def draw_auto_center_screen(
    color_image_bgr,
    box,
    stable_frame_count,
    failed_auto_moves,
    total_auto_moves,
):
    draw_auto_text(
        color_image_bgr,
        "AUTO CENTERING BEFORE SCAN",
        30,
        (0, 255, 255),
    )

    draw_auto_text(
        color_image_bgr,
        "S = start scan manually | H = home | C = center reference | Q = quit",
        60,
        (255, 255, 255),
    )

    draw_auto_text(
        color_image_bgr,
        f"Moves: {total_auto_moves}/{AUTO_MAX_TOTAL_MOVES} | Failed: {failed_auto_moves}/{AUTO_MAX_FAILED_MOVES}",
        90,
        (255, 255, 255),
    )

    if box is None:
        draw_auto_text(
            color_image_bgr,
            "No box detected",
            120,
            (0, 0, 255),
        )
        return

    draw_auto_box(color_image_bgr, box)

    offset_x, offset_y = get_auto_box_offset_pixels(box)
    centered_status = "Centered" if is_auto_box_centered(box) else "Moving"

    draw_auto_text(
        color_image_bgr,
        (
            f"Offset X={offset_x}px Y={offset_y}px | "
            f"{centered_status} | Stable {stable_frame_count}/{AUTO_REQUIRED_STABLE_FRAMES}"
        ),
        120,
        (0, 255, 0),
    )


def close_auto_windows():
    for window_name in [AUTO_WINDOW_NAME, AUTO_MASK_WINDOW_NAME]:
        try:
            cv2.destroyWindow(window_name)
        except cv2.error:
            pass


def auto_center_camera_on_box(
    robot,
    rdk,
    pipeline,
    align,
    depth_scale,
    T_tcp_camera,
    T_camera_tcp,
):
    previous_box = None
    stable_frame_count = 0
    failed_auto_moves = 0
    total_auto_moves = 0
    last_auto_move_time = 0.0
    start_time = time.time()
    last_print_time = 0.0

    print("")
    print("=" * 70)
    print("AUTO CENTERING STARTED")
    print("=" * 70)
    print("The robot will center the camera on the detected open box.")
    print("When centered, the code will continue with the reference capture.")
    print("Press S to skip centering and start the scan from the current pose.")
    print("=" * 70)

    while True:
        if time.time() - start_time > AUTO_CENTER_TIMEOUT_SECONDS:
            close_auto_windows()
            raise Exception("Auto centering timed out before the box was centered.")

        depth_frame, color_image_rgb, depth_image = get_aligned_realsense_frame(
            pipeline,
            align,
        )

        if depth_frame is None:
            continue

        color_image_bgr = cv2.cvtColor(color_image_rgb, cv2.COLOR_RGB2BGR)
        box, mask = detect_auto_box(depth_image, depth_scale)

        stable_frame_count, previous_box = update_auto_stability(
            box,
            previous_box,
            stable_frame_count,
        )

        draw_auto_center_screen(
            color_image_bgr,
            box,
            stable_frame_count,
            failed_auto_moves,
            total_auto_moves,
        )

        if box is not None and time.time() - last_print_time > 0.5:
            offset_x, offset_y = get_auto_box_offset_pixels(box)
            print(
                "Auto box:",
                f"center=({box['center_x']}, {box['center_y']}),",
                f"offset=({offset_x}, {offset_y}),",
                f"distance={box['distance_meters']:.2f}m,",
                f"stable={stable_frame_count}/{AUTO_REQUIRED_STABLE_FRAMES}",
            )
            last_print_time = time.time()

        if mask is not None:
            cv2.imshow(AUTO_MASK_WINDOW_NAME, mask)

        cv2.imshow(AUTO_WINDOW_NAME, color_image_bgr)

        key = cv2.waitKey(1) & 0xFF

        if key == ord("q") or key == 27:
            close_auto_windows()
            raise KeyboardInterrupt

        if key == ord("s"):
            print("")
            print("Manual skip selected. Starting scan from current robot pose.")
            close_auto_windows()
            return get_robot_joints_when_ready(robot)

        if key == ord("h"):
            failed_auto_moves = 0
            total_auto_moves = 0
            stable_frame_count = 0
            previous_box = None
            move_robot_to_joints(robot, rdk, HOME_JOINTS, "Home_From_Auto_Center")

        if key == ord("c"):
            failed_auto_moves = 0
            total_auto_moves = 0
            stable_frame_count = 0
            previous_box = None
            move_robot_to_joints(
                robot,
                rdk,
                CENTER_REFERENCE_JOINTS,
                "Center_Reference_From_Auto_Center",
            )

        if box is not None and is_auto_box_centered(box):
            if stable_frame_count >= AUTO_REQUIRED_STABLE_FRAMES:
                print("")
                print("=" * 70)
                print("AUTO CENTERING FINISHED")
                print("=" * 70)
                print("The camera is centered on the box.")
                print("Continuing with reference point cloud capture.")
                print("=" * 70)
                close_auto_windows()
                return get_robot_joints_when_ready(robot)

        if should_auto_center_move(
            box,
            stable_frame_count,
            last_auto_move_time,
            failed_auto_moves,
            total_auto_moves,
        ):
            point_camera = get_auto_box_center_3d(depth_frame, box)

            if point_camera is None:
                print("Auto move skipped. No valid 3D box center.")
                failed_auto_moves += 1
            else:
                actual_joints = move_camera_one_auto_step_to_box_center(
                    robot,
                    rdk,
                    T_tcp_camera,
                    T_camera_tcp,
                    point_camera,
                )

                if actual_joints is None:
                    failed_auto_moves += 1
                else:
                    failed_auto_moves = 0
                    total_auto_moves += 1

            stable_frame_count = 0
            previous_box = None
            last_auto_move_time = time.time()

        if failed_auto_moves >= AUTO_MAX_FAILED_MOVES:
            close_auto_windows()
            raise Exception("Auto centering stopped because too many robot moves failed.")

        if total_auto_moves >= AUTO_MAX_TOTAL_MOVES:
            close_auto_windows()
            raise Exception("Auto centering stopped because the maximum move count was reached.")



# ─────────────────────────────────────────────────────────────────────────────
# MAIN
# ─────────────────────────────────────────────────────────────────────────────

def main():
    OUTPUT_FOLDER.mkdir(parents=True, exist_ok=True)

    rdk = Robolink()
    robot = rdk.ItemUserPick("Select your Doosan M0609 robot", ITEM_TYPE_ROBOT)

    if not robot.Valid():
        raise Exception("No valid robot selected.")

    print("Selected robot:", robot.Name())

    connect_robot(robot, rdk)

    T_tcp_mount = xyzrxryrz_to_numpy(TCP_TO_CAMERA_MOUNT)
    T_mount_optical = xyzrxryrz_to_numpy(CAMERA_MOUNT_TO_OPTICAL)
    T_tcp_camera = T_tcp_mount @ T_mount_optical
    T_camera_tcp = np.linalg.inv(T_tcp_camera)

    print_transform("T_tcp_camera", T_tcp_camera)

    pipeline = None
    combined_point_cloud = o3d.geometry.PointCloud()

    successful_scans = 0
    skipped_scans = 0
    unsafe_scans = 0
    failed_moves = 0

    try:
        (
            pipeline,
            align,
            depth_scale,
            intrinsic_o3d,
            spatial_filter,
            temporal_filter,
            hole_filling_filter,
        ) = start_realsense()

        print("\n" + "=" * 70)
        print("AUTO-CENTERED ADAPTIVE INSIDE-BOX SCANNING STARTED")
        print("=" * 70)
        print("Step 1: Center the camera on the open box.")
        print("Step 2: Capture the reference scan from the centered pose.")
        print("Step 3: Generate adaptive scan poses.")
        print("Step 4: Capture and merge all scans.")
        print("=" * 70)

        if AUTO_CENTER_BEFORE_SCAN:
            center_actual_joints = auto_center_camera_on_box(
                robot,
                rdk,
                pipeline,
                align,
                depth_scale,
                T_tcp_camera,
                T_camera_tcp,
            )
        else:
            center_actual_joints = move_robot_to_joints(
                robot,
                rdk,
                CENTER_REFERENCE_JOINTS,
                "Cabinet_Center_Reference",
            )

        T_base_tcp_center = robodk_mat_to_numpy(robot.SolveFK(center_actual_joints))
        T_base_camera_center = T_base_tcp_center @ T_tcp_camera

        print_transform("T_base_tcp_center", T_base_tcp_center)
        print_transform("T_base_camera_center", T_base_camera_center)

        reference_cloud = capture_stable_pointcloud(
            pipeline,
            align,
            intrinsic_o3d,
            depth_scale,
            spatial_filter,
            temporal_filter,
            hole_filling_filter,
            CAPTURE_FRAMES_PER_POSITION,
        )

        if reference_cloud is None:
            raise Exception("Reference scan failed. No point cloud was captured.")

        print_cloud_bounds("Reference raw camera-frame scan", reference_cloud)
        adaptive_bounds = estimate_camera_cloud_bounds(reference_cloud)

        reference_cloud_cropped = crop_pointcloud_adaptive(
            reference_cloud,
            adaptive_bounds,
        )

        reference_cloud_cropped.transform(T_base_camera_center)
        reference_clean_scan = clean_pointcloud(reference_cloud_cropped)

        if len(reference_clean_scan.points) > 0:
            save_debug_scan("Reference_Center", reference_clean_scan)
            combined_point_cloud += reference_clean_scan
            successful_scans += 1
            print(
                f"Accepted scan {successful_scans}: Reference_Center "
                f"with {len(reference_clean_scan.points):,} cleaned points"
            )
        else:
            print("WARNING: Reference scan became empty after cleaning.")
            skipped_scans += 1

        generated_camera_poses = generate_scan_camera_poses_from_center(
            T_base_camera_center,
            adaptive_bounds,
        )

        for label, T_base_camera_target in generated_camera_poses:
            if label == "Reference_Center":
                continue

            T_base_tcp_target = T_base_camera_target @ T_camera_tcp

            if not is_generated_pose_safe(
                T_base_tcp_target,
                T_base_camera_target,
                label,
            ):
                unsafe_scans += 1
                skipped_scans += 1
                continue

            try:
                actual_joints = move_robot_to_pose(
                    robot,
                    rdk,
                    T_base_tcp_target,
                    label,
                )
            except Exception as error:
                print("")
                print(f"WARNING: Could not move to generated pose {label}.")
                print("Move error:", error)
                failed_moves += 1
                skipped_scans += 1
                continue

            T_base_tcp_actual = robodk_mat_to_numpy(robot.SolveFK(actual_joints))
            T_base_camera_actual = T_base_tcp_actual @ T_tcp_camera

            print_transform(f"T_base_tcp_actual_{label}", T_base_tcp_actual)
            print_transform(f"T_base_camera_actual_{label}", T_base_camera_actual)

            clean_scan = scan_current_position(
                label,
                pipeline,
                align,
                intrinsic_o3d,
                depth_scale,
                spatial_filter,
                temporal_filter,
                hole_filling_filter,
                T_base_camera_actual,
                adaptive_bounds,
            )

            if clean_scan is None:
                skipped_scans += 1
                continue

            combined_point_cloud += clean_scan
            successful_scans += 1

            print(
                f"Accepted scan {successful_scans}: {label} "
                f"with {len(clean_scan.points):,} cleaned points"
            )

    except KeyboardInterrupt:
        print("\nScanning interrupted by user.")

    finally:
        if pipeline is not None:
            pipeline.stop()
            print("\nRealSense stopped.")

        cv2.destroyAllWindows()

        try:
            move_robot_to_joints(
                robot,
                rdk,
                HOME_JOINTS,
                "Home_End",
            )
        except Exception as error:
            print("Could not move robot back to home position:", error)

    print("\n" + "=" * 70)
    print("SCAN SUMMARY")
    print("=" * 70)
    print("Successful scans:", successful_scans)
    print("Skipped scans:", skipped_scans)
    print("Unsafe skipped scans:", unsafe_scans)
    print("Failed robot moves:", failed_moves)
    print("Total merged points before final cleanup:", len(combined_point_cloud.points))
    print_cloud_bounds("Combined point cloud before final cleanup", combined_point_cloud)

    if len(combined_point_cloud.points) == 0:
        raise Exception("No valid point cloud was captured. Combined cloud is empty.")

    combined_point_cloud = clean_pointcloud(combined_point_cloud)
    combined_point_cloud = estimate_normals(combined_point_cloud)

    print("Total merged points after final cleanup:", len(combined_point_cloud.points))
    print_cloud_bounds("Combined point cloud after final cleanup", combined_point_cloud)

    o3d.io.write_point_cloud(str(OUTPUT_CLEAN_FILE), combined_point_cloud)
    print("Saved final merged point cloud to:", OUTPUT_CLEAN_FILE)

    if SHOW_FINAL_CLOUD:
        o3d.visualization.draw_geometries(
            [combined_point_cloud],
            window_name=f"Adaptive Inside Box Point Cloud - {successful_scans} scans",
        )

    print("Done.")


if __name__ == "__main__":
    main()

--- Python program Prog6 ---
import sys
import time
import math

import cv2
import numpy as np
import pyrealsense2 as rs

sys.path.append("C:/RoboDK/Python")

from robodk.robolink import *
from robodk.robomath import TxyzRxyz_2_Pose, Mat


# =============================================================================
# CONFIGURATION
# =============================================================================

RUN_ON_REAL_ROBOT = True

AUTO_MOVE_ENABLED = True
MOVE_TO_CENTER_REFERENCE_ON_START = False

HOME_JOINTS = [270.00, 0.00, 90.00, 180.00, 0.00, 0.00]
CENTER_REFERENCE_JOINTS = [270.01, 0.21, 98.95, 180.00, 6.92, 0.00]

TCP_TO_CAMERA_MOUNT = [0, 0, 55, 0, 0, 0]
CAMERA_MOUNT_TO_OPTICAL = [0, 0, 0, 0, 0, 90]

COLOR_WIDTH = 640
COLOR_HEIGHT = 480
FPS = 30

MIN_DEPTH_METERS = 0.20
MAX_DEPTH_METERS = 3.00
TARGET_DISTANCE_METERS = 0.90

MAX_TRANSLATION_STEP_METERS = 0.025
CENTERING_GAIN = 0.60
DEPTH_GAIN = 0.60

CENTER_TOLERANCE_PIXELS = 25
DISTANCE_TOLERANCE_METERS = 0.05

REQUIRED_STABLE_FRAMES = 8
STABLE_CENTER_TOLERANCE_PIXELS = 12
STABLE_DISTANCE_TOLERANCE_METERS = 0.04
AUTO_MOVE_COOLDOWN_SECONDS = 1.25
MAX_FAILED_AUTO_MOVES = 5

MIN_BOX_AREA = 1200
MIN_BOX_WIDTH = 80
MIN_BOX_HEIGHT = 80

DEPTH_PERCENTILE = 10
DEPTH_FRONT_MARGIN = 0.05
DEPTH_BACK_MARGIN = 0.45

DETECTION_ROI_TOP_RATIO = 0.05
DETECTION_ROI_BOTTOM_RATIO = 0.82
DETECTION_ROI_LEFT_RATIO = 0.02
DETECTION_ROI_RIGHT_RATIO = 0.98

MIN_SAFE_TCP_Z_MM = 120.0
MIN_SAFE_CAMERA_Z_MM = 120.0

SETTLE_TIME = 0.75
MOVE_TIMEOUT_SEC = 30.0
POLL_INTERVAL_SEC = 0.1

WINDOW_NAME = "Automatic Box Centering"
MASK_WINDOW_NAME = "Depth Mask"


# =============================================================================
# MATRIX HELPERS
# =============================================================================

def robodk_mat_to_numpy(mat):
    transform = np.eye(4, dtype=np.float64)

    for row in range(3):
        for col in range(3):
            transform[row, col] = mat[row, col]

        transform[row, 3] = mat[row, 3] / 1000.0

    return transform


def numpy_to_robodk_mat(transform):
    return Mat([
        [
            transform[0, 0],
            transform[0, 1],
            transform[0, 2],
            transform[0, 3] * 1000.0,
        ],
        [
            transform[1, 0],
            transform[1, 1],
            transform[1, 2],
            transform[1, 3] * 1000.0,
        ],
        [
            transform[2, 0],
            transform[2, 1],
            transform[2, 2],
            transform[2, 3] * 1000.0,
        ],
        [0, 0, 0, 1],
    ])


def xyzrxryrz_to_numpy(pose_values):
    pose = TxyzRxyz_2_Pose([
        pose_values[0],
        pose_values[1],
        pose_values[2],
        math.radians(pose_values[3]),
        math.radians(pose_values[4]),
        math.radians(pose_values[5]),
    ])

    return robodk_mat_to_numpy(pose)


def make_local_offset_transform(offset_x, offset_y, offset_z):
    transform = np.eye(4, dtype=np.float64)

    transform[0, 3] = offset_x
    transform[1, 3] = offset_y
    transform[2, 3] = offset_z

    return transform


def joints_to_list(joints_mat):
    try:
        return list(joints_mat.list())
    except Exception:
        try:
            return list(joints_mat)
        except Exception:
            return [joints_mat[index] for index in range(len(joints_mat))]


# =============================================================================
# ROBOT HELPERS
# =============================================================================

def connect_robot(robot, rdk):
    if RUN_ON_REAL_ROBOT:
        rdk.setRunMode(RUNMODE_RUN_ROBOT)

        status = robot.ConnectSafe()
        print("ConnectSafe status:", status)

        if status != ROBOTCOM_READY:
            raise Exception("Robot is not ready. Check RoboDK connection settings.")
    else:
        rdk.setRunMode(RUNMODE_SIMULATE)
        print("Running in RoboDK simulation mode.")


def wait_until_robot_stops(robot, timeout_sec=MOVE_TIMEOUT_SEC):
    start = time.time()

    while True:
        try:
            if not robot.Busy():
                return
        except Exception:
            pass

        if time.time() - start > timeout_sec:
            raise Exception("Timeout waiting for robot to stop.")

        time.sleep(POLL_INTERVAL_SEC)


def get_robot_joints_when_ready(robot, timeout_sec=5.0):
    start = time.time()

    while True:
        try:
            return joints_to_list(robot.Joints())
        except Exception:
            if time.time() - start > timeout_sec:
                raise Exception("Could not read robot joints.")

            time.sleep(POLL_INTERVAL_SEC)


def move_robot_to_joints(robot, rdk, joints, label):
    target = rdk.AddTarget(f"_auto_box_{label}")
    target.setAsJointTarget()
    target.setJoints(joints)

    print("")
    print(f"Moving to {label}: {[round(joint, 2) for joint in joints]}")

    if RUN_ON_REAL_ROBOT:
        rdk.setRunMode(RUNMODE_RUN_ROBOT)
    else:
        rdk.setRunMode(RUNMODE_SIMULATE)

    robot.MoveJ(target, blocking=False)
    wait_until_robot_stops(robot)

    target.Delete()

    print(f"Arrived at {label}. Settling for {SETTLE_TIME:.1f} seconds...")
    time.sleep(SETTLE_TIME)

    return get_robot_joints_when_ready(robot)


def move_robot_to_pose(robot, rdk, T_base_tcp, label):
    target = rdk.AddTarget(f"_auto_box_{label}")
    target_pose = numpy_to_robodk_mat(T_base_tcp)

    target.setPose(target_pose)
    target.setAsCartesianTarget()

    print("")
    print(f"Moving to generated pose: {label}")
    print(f"Target TCP X: {T_base_tcp[0, 3] * 1000.0:.1f} mm")
    print(f"Target TCP Y: {T_base_tcp[1, 3] * 1000.0:.1f} mm")
    print(f"Target TCP Z: {T_base_tcp[2, 3] * 1000.0:.1f} mm")

    if RUN_ON_REAL_ROBOT:
        rdk.setRunMode(RUNMODE_RUN_ROBOT)
    else:
        rdk.setRunMode(RUNMODE_SIMULATE)

    robot.MoveJ(target, blocking=False)
    wait_until_robot_stops(robot)

    target.Delete()

    print(f"Arrived at {label}. Settling for {SETTLE_TIME:.1f} seconds...")
    time.sleep(SETTLE_TIME)

    return get_robot_joints_when_ready(robot)


def is_generated_pose_safe(T_base_tcp, T_base_camera, label):
    tcp_z_mm = T_base_tcp[2, 3] * 1000.0
    camera_z_mm = T_base_camera[2, 3] * 1000.0

    if tcp_z_mm < MIN_SAFE_TCP_Z_MM:
        print("")
        print(f"SKIPPING {label}")
        print(f"Reason: TCP Z is too low: {tcp_z_mm:.1f} mm")
        return False

    if camera_z_mm < MIN_SAFE_CAMERA_Z_MM:
        print("")
        print(f"SKIPPING {label}")
        print(f"Reason: Camera Z is too low: {camera_z_mm:.1f} mm")
        return False

    return True


def calculate_camera_correction(point_camera):
    camera_offset = np.array([
        point_camera[0] * CENTERING_GAIN,
        point_camera[1] * CENTERING_GAIN,
        (point_camera[2] - TARGET_DISTANCE_METERS) * DEPTH_GAIN,
    ])

    offset_size = np.linalg.norm(camera_offset)

    if offset_size > MAX_TRANSLATION_STEP_METERS:
        camera_offset = (
            camera_offset / offset_size
        ) * MAX_TRANSLATION_STEP_METERS

    return camera_offset


def move_camera_one_step_to_box_center(
    robot,
    rdk,
    T_tcp_camera,
    T_camera_tcp,
    point_camera,
):
    actual_joints = get_robot_joints_when_ready(robot)

    T_base_tcp_current = robodk_mat_to_numpy(robot.SolveFK(actual_joints))
    T_base_camera_current = T_base_tcp_current @ T_tcp_camera

    camera_offset = calculate_camera_correction(point_camera)

    T_camera_offset = make_local_offset_transform(
        camera_offset[0],
        camera_offset[1],
        camera_offset[2],
    )

    T_base_camera_target = T_base_camera_current @ T_camera_offset
    T_base_tcp_target = T_base_camera_target @ T_camera_tcp

    print("")
    print("Automatic box-centering movement")
    print("3D box point in camera frame:", np.round(point_camera, 4), "m")
    print("Camera movement step:", np.round(camera_offset, 4), "m")
    print("Current robot joints:", [round(joint, 2) for joint in actual_joints])

    if not is_generated_pose_safe(
        T_base_tcp_target,
        T_base_camera_target,
        "Auto_Box_Center_Step",
    ):
        return None

    try:
        return move_robot_to_pose(
            robot,
            rdk,
            T_base_tcp_target,
            "Auto_Box_Center_Step",
        )
    except Exception as error:
        print("")
        print("Could not move robot to automatic box center step.")
        print("Move error:", error)
        return None


# =============================================================================
# REALSENSE HELPERS
# =============================================================================

def start_realsense():
    print("")
    print("Starting Intel RealSense camera...")

    pipeline = rs.pipeline()
    config = rs.config()

    config.enable_stream(
        rs.stream.color,
        COLOR_WIDTH,
        COLOR_HEIGHT,
        rs.format.bgr8,
        FPS,
    )

    config.enable_stream(
        rs.stream.depth,
        COLOR_WIDTH,
        COLOR_HEIGHT,
        rs.format.z16,
        FPS,
    )

    profile = pipeline.start(config)
    depth_sensor = profile.get_device().first_depth_sensor()

    if depth_sensor.supports(rs.option.visual_preset):
        try:
            depth_sensor.set_option(
                rs.option.visual_preset,
                int(rs.rs400_visual_preset.high_density),
            )
            print("Visual preset: HIGH_DENSITY")
        except Exception as error:
            print("Could not set HIGH_DENSITY preset:", error)

    if depth_sensor.supports(rs.option.emitter_enabled):
        try:
            depth_sensor.set_option(rs.option.emitter_enabled, 1)
            print("Emitter enabled.")
        except Exception as error:
            print("Could not enable emitter:", error)

    if depth_sensor.supports(rs.option.laser_power):
        try:
            laser_range = depth_sensor.get_option_range(rs.option.laser_power)
            depth_sensor.set_option(rs.option.laser_power, laser_range.max)
            print("Laser power set to max:", laser_range.max)
        except Exception as error:
            print("Could not set laser power:", error)

    depth_scale = depth_sensor.get_depth_scale()
    align = rs.align(rs.stream.color)

    print("RealSense ready.")
    print("Depth scale:", depth_scale)

    return pipeline, align, depth_scale


def get_camera_frame(pipeline, align):
    frames = pipeline.wait_for_frames()
    aligned_frames = align.process(frames)

    color_frame = aligned_frames.get_color_frame()
    depth_frame = aligned_frames.get_depth_frame()

    if not color_frame or not depth_frame:
        return None, None, None

    color_image = np.asanyarray(color_frame.get_data())
    depth_image = np.asanyarray(depth_frame.get_data())

    return depth_frame, color_image, depth_image


# =============================================================================
# BOX DETECTION
# =============================================================================

def get_depth_in_region(depth_image, depth_scale, x1, y1, x2, y2):
    image_height, image_width = depth_image.shape

    x1 = max(0, min(int(x1), image_width))
    x2 = max(0, min(int(x2), image_width))
    y1 = max(0, min(int(y1), image_height))
    y2 = max(0, min(int(y2), image_height))

    if x2 <= x1 or y2 <= y1:
        return None

    depth_crop = depth_image[y1:y2, x1:x2].astype(np.float32) * depth_scale

    valid_depth = depth_crop[
        (depth_crop > MIN_DEPTH_METERS)
        & (depth_crop < MAX_DEPTH_METERS)
    ]

    if valid_depth.size == 0:
        return None

    return float(np.percentile(valid_depth, 30))


def create_detection_roi_mask(image_height, image_width):
    roi_mask = np.zeros((image_height, image_width), dtype=np.uint8)

    x1 = int(image_width * DETECTION_ROI_LEFT_RATIO)
    x2 = int(image_width * DETECTION_ROI_RIGHT_RATIO)
    y1 = int(image_height * DETECTION_ROI_TOP_RATIO)
    y2 = int(image_height * DETECTION_ROI_BOTTOM_RATIO)

    roi_mask[y1:y2, x1:x2] = 255

    return roi_mask


def create_depth_mask(depth_image, depth_scale):
    image_height, image_width = depth_image.shape
    depth_meters = depth_image.astype(np.float32) * depth_scale

    roi_mask = create_detection_roi_mask(image_height, image_width)

    valid_mask = (
        (depth_meters > MIN_DEPTH_METERS)
        & (depth_meters < MAX_DEPTH_METERS)
        & (roi_mask == 255)
    )

    if not np.any(valid_mask):
        return None

    valid_depth_values = depth_meters[valid_mask]

    front_depth = np.percentile(
        valid_depth_values,
        DEPTH_PERCENTILE,
    )

    mask = (
        valid_mask
        & (depth_meters > front_depth - DEPTH_FRONT_MARGIN)
        & (depth_meters < front_depth + DEPTH_BACK_MARGIN)
    )

    mask = mask.astype(np.uint8) * 255

    close_kernel = np.ones((11, 11), np.uint8)
    open_kernel = np.ones((5, 5), np.uint8)

    mask = cv2.morphologyEx(
        mask,
        cv2.MORPH_CLOSE,
        close_kernel,
        iterations=3,
    )

    mask = cv2.morphologyEx(
        mask,
        cv2.MORPH_OPEN,
        open_kernel,
        iterations=1,
    )

    mask = cv2.bitwise_and(mask, roi_mask)

    return mask


def detect_box(depth_image, depth_scale):
    mask = create_depth_mask(depth_image, depth_scale)

    if mask is None:
        return None, None

    contours, _ = cv2.findContours(
        mask,
        cv2.RETR_EXTERNAL,
        cv2.CHAIN_APPROX_SIMPLE,
    )

    image_height, image_width = depth_image.shape
    image_center_x = image_width / 2.0
    image_center_y = image_height / 2.0

    best_box = None
    best_score = 0

    for contour in contours:
        area = cv2.contourArea(contour)

        if area < MIN_BOX_AREA:
            continue

        x, y, width, height = cv2.boundingRect(contour)

        if width < MIN_BOX_WIDTH or height < MIN_BOX_HEIGHT:
            continue

        if width > image_width * 0.98 or height > image_height * 0.98:
            continue

        aspect_ratio = width / float(height)

        if aspect_ratio < 0.50 or aspect_ratio > 4.50:
            continue

        x1 = x
        y1 = y
        x2 = x + width
        y2 = y + height

        center_x = int((x1 + x2) / 2)
        center_y = int((y1 + y2) / 2)

        distance_meters = get_depth_in_region(
            depth_image,
            depth_scale,
            x1,
            y1,
            x2,
            y2,
        )

        if distance_meters is None:
            continue

        center_error = np.sqrt(
            (center_x - image_center_x) ** 2
            + (center_y - image_center_y) ** 2
        )

        area_score = area / float(image_width * image_height)
        center_score = 1.0 / (1.0 + center_error)

        score = area_score * 1000.0 + center_score * 150.0

        if score > best_score:
            best_score = score

            best_box = {
                "source": "depth_rectangle",
                "x1": x1,
                "y1": y1,
                "x2": x2,
                "y2": y2,
                "center_x": center_x,
                "center_y": center_y,
                "distance_meters": distance_meters,
                "area": area,
            }

    return best_box, mask


def get_box_center_3d(depth_frame, box):
    center_x = box["center_x"]
    center_y = box["center_y"]
    depth_meters = box["distance_meters"]

    if depth_meters is None:
        return None

    if depth_meters <= MIN_DEPTH_METERS or depth_meters >= MAX_DEPTH_METERS:
        return None

    intrinsics = depth_frame.profile.as_video_stream_profile().intrinsics

    point_camera = rs.rs2_deproject_pixel_to_point(
        intrinsics,
        [center_x, center_y],
        depth_meters,
    )

    return np.array(point_camera, dtype=np.float64)


# =============================================================================
# AUTO CENTERING LOGIC
# =============================================================================

def get_box_offset_pixels(box):
    image_center_x = int(COLOR_WIDTH / 2)
    image_center_y = int(COLOR_HEIGHT / 2)

    offset_x = box["center_x"] - image_center_x
    offset_y = box["center_y"] - image_center_y

    return offset_x, offset_y


def is_box_centered(box):
    offset_x, offset_y = get_box_offset_pixels(box)

    center_error = np.sqrt(offset_x ** 2 + offset_y ** 2)
    distance_error = abs(box["distance_meters"] - TARGET_DISTANCE_METERS)

    return (
        center_error <= CENTER_TOLERANCE_PIXELS
        and distance_error <= DISTANCE_TOLERANCE_METERS
    )


def is_box_stable(current_box, previous_box):
    if current_box is None or previous_box is None:
        return False

    center_change = np.sqrt(
        (current_box["center_x"] - previous_box["center_x"]) ** 2
        + (current_box["center_y"] - previous_box["center_y"]) ** 2
    )

    distance_change = abs(
        current_box["distance_meters"] - previous_box["distance_meters"]
    )

    return (
        center_change <= STABLE_CENTER_TOLERANCE_PIXELS
        and distance_change <= STABLE_DISTANCE_TOLERANCE_METERS
    )


def update_stability(box, previous_box, stable_frame_count):
    if box is None:
        return 0, None

    if is_box_stable(box, previous_box):
        stable_frame_count += 1
    else:
        stable_frame_count = 1

    return stable_frame_count, box


def should_auto_move(
    box,
    stable_frame_count,
    last_auto_move_time,
    failed_auto_moves,
):
    if not AUTO_MOVE_ENABLED:
        return False

    if box is None:
        return False

    if is_box_centered(box):
        return False

    if stable_frame_count < REQUIRED_STABLE_FRAMES:
        return False

    if time.time() - last_auto_move_time < AUTO_MOVE_COOLDOWN_SECONDS:
        return False

    if failed_auto_moves >= MAX_FAILED_AUTO_MOVES:
        return False

    return True


# =============================================================================
# DRAWING
# =============================================================================

def draw_box(image, box):
    image_center_x = int(COLOR_WIDTH / 2)
    image_center_y = int(COLOR_HEIGHT / 2)

    cv2.rectangle(
        image,
        (box["x1"], box["y1"]),
        (box["x2"], box["y2"]),
        (0, 255, 0),
        3,
    )

    cv2.circle(
        image,
        (box["center_x"], box["center_y"]),
        7,
        (0, 0, 255),
        -1,
    )

    cv2.line(
        image,
        (image_center_x - 15, image_center_y),
        (image_center_x + 15, image_center_y),
        (255, 0, 0),
        2,
    )

    cv2.line(
        image,
        (image_center_x, image_center_y - 15),
        (image_center_x, image_center_y + 15),
        (255, 0, 0),
        2,
    )

    cv2.line(
        image,
        (image_center_x, image_center_y),
        (box["center_x"], box["center_y"]),
        (0, 255, 255),
        2,
    )

    cv2.putText(
        image,
        f"Box | {box['distance_meters']:.2f} m",
        (box["x1"], max(box["y1"] - 10, 25)),
        cv2.FONT_HERSHEY_SIMPLEX,
        0.65,
        (0, 255, 0),
        2,
    )


def draw_text(image, text, y, color):
    cv2.putText(
        image,
        text,
        (10, y),
        cv2.FONT_HERSHEY_SIMPLEX,
        0.65,
        color,
        2,
    )


def draw_screen(
    color_image,
    box,
    fps,
    stable_frame_count,
    failed_auto_moves,
):
    draw_text(
        color_image,
        f"FPS: {fps:.1f}",
        30,
        (255, 255, 255),
    )

    draw_text(
        color_image,
        "AUTO CENTERING ENABLED",
        60,
        (0, 255, 255),
    )

    draw_text(
        color_image,
        "C = center reference | H = home | Q = quit",
        90,
        (255, 255, 255),
    )

    if failed_auto_moves >= MAX_FAILED_AUTO_MOVES:
        draw_text(
            color_image,
            "AUTO STOPPED: too many failed moves",
            120,
            (0, 0, 255),
        )
        return

    if box is None:
        draw_text(
            color_image,
            "No box detected",
            120,
            (0, 0, 255),
        )
        return

    draw_box(color_image, box)

    offset_x, offset_y = get_box_offset_pixels(box)

    centered_status = "Centered" if is_box_centered(box) else "Moving"

    draw_text(
        color_image,
        (
            f"Offset X={offset_x}px Y={offset_y}px | "
            f"{centered_status} | Stable {stable_frame_count}/{REQUIRED_STABLE_FRAMES}"
        ),
        120,
        (0, 255, 0),
    )


# =============================================================================
# MAIN
# =============================================================================

def main():
    rdk = Robolink()

    robot = rdk.ItemUserPick(
        "Select your Doosan M0609 robot",
        ITEM_TYPE_ROBOT,
    )

    if not robot.Valid():
        raise Exception("No valid robot selected.")

    print("Selected robot:", robot.Name())

    connect_robot(robot, rdk)

    T_tcp_mount = xyzrxryrz_to_numpy(TCP_TO_CAMERA_MOUNT)
    T_mount_optical = xyzrxryrz_to_numpy(CAMERA_MOUNT_TO_OPTICAL)

    T_tcp_camera = T_tcp_mount @ T_mount_optical
    T_camera_tcp = np.linalg.inv(T_tcp_camera)

    pipeline = None

    previous_box = None
    stable_frame_count = 0
    last_auto_move_time = 0.0
    failed_auto_moves = 0

    previous_time = time.time()
    last_print_time = 0.0

    try:
        if MOVE_TO_CENTER_REFERENCE_ON_START:
            move_robot_to_joints(
                robot,
                rdk,
                CENTER_REFERENCE_JOINTS,
                "Center_Reference_Start",
            )

        pipeline, align, depth_scale = start_realsense()

        while True:
            depth_frame, color_image, depth_image = get_camera_frame(
                pipeline,
                align,
            )

            if depth_frame is None:
                continue

            box, mask = detect_box(depth_image, depth_scale)

            stable_frame_count, previous_box = update_stability(
                box,
                previous_box,
                stable_frame_count,
            )

            current_time = time.time()
            fps = 1.0 / max(current_time - previous_time, 0.0001)
            previous_time = current_time

            draw_screen(
                color_image,
                box,
                fps,
                stable_frame_count,
                failed_auto_moves,
            )

            if current_time - last_print_time > 0.5 and box is not None:
                offset_x, offset_y = get_box_offset_pixels(box)

                print(
                    "Box:",
                    f"x1={box['x1']},",
                    f"y1={box['y1']},",
                    f"x2={box['x2']},",
                    f"y2={box['y2']},",
                    f"center=({box['center_x']}, {box['center_y']}),",
                    f"offset=({offset_x}, {offset_y}),",
                    f"distance={box['distance_meters']:.2f}m,",
                    f"stable={stable_frame_count}/{REQUIRED_STABLE_FRAMES}",
                )

                last_print_time = current_time

            if mask is not None:
                cv2.imshow(MASK_WINDOW_NAME, mask)

            cv2.imshow(WINDOW_NAME, color_image)

            if should_auto_move(
                box,
                stable_frame_count,
                last_auto_move_time,
                failed_auto_moves,
            ):
                point_camera = get_box_center_3d(depth_frame, box)

                if point_camera is None:
                    print("Auto move skipped. No valid 3D box center.")
                    failed_auto_moves += 1
                else:
                    actual_joints = move_camera_one_step_to_box_center(
                        robot,
                        rdk,
                        T_tcp_camera,
                        T_camera_tcp,
                        point_camera,
                    )

                    if actual_joints is None:
                        failed_auto_moves += 1
                    else:
                        failed_auto_moves = 0

                stable_frame_count = 0
                previous_box = None
                last_auto_move_time = time.time()

            key = cv2.waitKey(1) & 0xFF

            if key == ord("q") or key == 27:
                break

            if key == ord("h"):
                failed_auto_moves = 0
                stable_frame_count = 0
                previous_box = None

                move_robot_to_joints(
                    robot,
                    rdk,
                    HOME_JOINTS,
                    "Home",
                )

            if key == ord("c"):
                failed_auto_moves = 0
                stable_frame_count = 0
                previous_box = None

                move_robot_to_joints(
                    robot,
                    rdk,
                    CENTER_REFERENCE_JOINTS,
                    "Center_Reference",
                )

    except KeyboardInterrupt:
        print("")
        print("Stopped by user.")

    finally:
        if pipeline is not None:
            pipeline.stop()
            print("RealSense stopped.")

        cv2.destroyAllWindows()
        print("Done.")


if __name__ == "__main__":
    main()
